FUNCTION TryConvert_LREAL_TO_UDINT : BOOL
VAR_INPUT
	in : LREAL;
	out : REFERENCE TO UDINT;
END_VAR

IF in > DatatypeLimits.MAX_VALUE_OF_LREAL_WHICH_CAN_BE_HELD_IN_A_UDINT THEN
	RETURN;
END_IF

IF in < DatatypeLimits.MIN_VALUE_OF_LREAL_WHICH_CAN_BE_HELD_IN_A_UDINT THEN
	RETURN;
END_IF

out := LREAL_TO_UDINT(in);
TryConvert_LREAL_TO_UDINT := TRUE;

END_FUNCTION

(* stored: Version 1.1.0.1, ProductVersion 3.1.4024.12
   POU TryConvert_LREAL_TO_UDINT: Id {d8f427f0-8d63-47e3-98f2-a25650992443}, SpecialFunc None *)
